// TIA Portal V21 export
TYPE "Priorità"
   STRUCT
      Soglia : Real;
      Isteresi : Real;
   END_STRUCT;
END_TYPE
